% RSLogix 500 project JOB 8.RSS, saved by version 10.00.00.00 %
PROJECT "UNTITLED"    % processor: Bul.1763 MicroLogix 1100 Series B %

PROGRAM FILES
  LAD 2   4 rungs

DATA FILES
  O0 OUTPUT  4 elements
  I1 INPUT  6 elements
  S2 STATUS  66 elements
  B3 BINARY  1 elements
  T4 TIMER  1 elements
  C5 COUNTER  1 elements
  R6 CONTROL  1 elements
  N7 INTEGER  1 elements
  F8 FLOAT  1 elements

LADDER 2
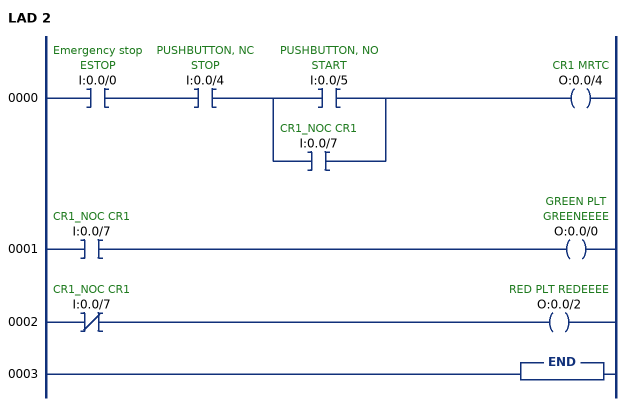
% Rung: 0 %  % edit flag set %
SOR XIC I:0.0/0 XIC I:0.0/4 BST XIC I:0.0/5 NXB XIC I:0.0/7 BND OTE O:0.0/4 EOR
%   I:0.0/0  ESTOP  "Emergency stop" %
%   I:0.0/4  STOP  "PUSHBUTTON, NC" %
%   I:0.0/5  START  "PUSHBUTTON, NO" %
%   I:0.0/7  CR1  "CR1_NOC" %
%   O:0.0/4  MRTC  "CR1" %
% Rung: 1 %  % edit flag set %
SOR XIC I:0.0/7 OTE O:0.0/0 EOR
%   I:0.0/7  CR1  "CR1_NOC" %
%   O:0.0/0  GREENEEEE  "GREEN PLT" %
% Rung: 2 %  % edit flag set %
SOR XIO I:0.0/7 OTE O:0.0/2 EOR
%   I:0.0/7  CR1  "CR1_NOC" %
%   O:0.0/2  REDEEEE  "RED PLT" %
% Rung: 3 %
SOR END EOR

OTHER DOCUMENTED ADDRESSES
  I:0.0/1  FWD  "Three position selector switch position A"
  I:0.0/2  REV  "Three Postion Selector Switch Postion B"
  I:0.0/3  RUN_JOG  "2 POS SLCT SWITCH"
  I:0.0/6  RJ  "PUSHBUTTON, NO"
  I:0.0/8  CR2_NOC  "CR2 NOC"
  I:0.0/9  REV_MTR_SRT_NOC  "REV MTR STARTER NOC"
  I:0.0/10  GREENIE  "GREEN PLT"
  I:0.0/11  YELLEEE  "YELLOW PLT"
  I:0.0/12  REDEEE  "RED PLT"
  I:0.0/13  BLUEEE  "BLUE PLT"
  I:0.0/14  MTR  "CR1 COIL 1"
  I:0.0/15  CR2_COIL_2  "CR2 COIL"
